// TIA Portal V18 export
DATA_BLOCK "dbDataFromMainPrg"   // DB3
{ S7_Optimized_Access := 'TRUE' }
// stored: MemoryReserve 100
   VAR
      tag1 : Bool;
      "tag2 TOTO" : Bool;
      tag3 : Bool;
      tag4 : UDInt;
      tag5 : Bool;
      tag6 : Bool;
      tag74 : Bool;
   END_VAR
BEGIN
END_DATA_BLOCK
